{attribute 'qualified_only'}
VAR_GLOBAL
END_VAR

(* stored: Version 1.1.0.1, ProductVersion 3.1.4022.7
   GVL GVL_03_Delay_Output: Id {0895c097-7662-4f11-b5fc-e03f894ba122} *)
